FUNCTION_BLOCK POU
VAR_INPUT
END_VAR
VAR_OUTPUT
END_VAR
VAR
END_VAR

END_FUNCTION_BLOCK

(* stored: Version 1.1.0.1, ProductVersion 3.1.4024.12
   POU POU: Id {00804c37-f8d2-4f16-9df0-e0fbf4f5ade9}, SpecialFunc None *)
